{attribute 'qualified_only'}
VAR_GLOBAL
END_VAR

(* stored: Version 1.1.0.1, ProductVersion 3.1.4022.12
   GVL GVL: Id {1281ad4e-62af-4abb-940f-db97be1f04b9} *)
